TYPE ST_TestCaseResult :
STRUCT
    TestName : Tc2_System.T_MaxString;
    TestClassName : Tc2_System.T_MaxString;
    TestIsFailed : BOOL;
    TestIsSkipped : BOOL;
    FailureMessage : Tc2_System.T_MaxString;
    FailureType : E_AssertionType;
    NumberOfAsserts : UINT;
    Duration : LREAL; // in seconds
END_STRUCT
END_TYPE

(* stored: Version 1.1.0.1, ProductVersion 3.1.4022.18
   DUT ST_TestCaseResult: Id {9c511c0b-2edf-4938-bd37-33f5b59a1386} *)
